// TIA Portal V21 export
TYPE "OBJ_IODevice_OUT_SICK_AFM60_Tel81_V105_Type"
   STRUCT
      STW2_ENC : Word;   // Encoder Control Word 2
      G1_STW : Word;   // Encoder Control Word 1
   END_STRUCT;
END_TYPE
